// TIA Portal V17 export
// export: Created 2025-03-20T13:42:24.3273325Z, ExportSetting WithDefaults, DisplayName Totally Integrated Automation Portal, DisplayVersion V17 Update 8, DisplayName TIA Portal Openness, DisplayVersion V17 Update 8, DisplayName TIA Portal Version Control Interface, DisplayVersion V17, DisplayName SINAMICS Startdrive Advanced, DisplayVersion V17 SP2, DisplayName SINAMICS Startdrive G110M, G120, G120C, G120D, G120P, G115D, DisplayVersion V17 SP2, DisplayName SINAMICS Startdrive G130, G150, S120, S150, SINAMICS MV, S210, DisplayVersion V17 SP2, DisplayName STEP 7 Professional, DisplayVersion V17 Update 8, DisplayName SINUMERIK ONE STEP 7 Toolbox, DisplayVersion V17 Update 12, DisplayName SINUMERIK 840D sl STEP 7 Toolbox, DisplayVersion V17 Update 12, DisplayName STEP 7 Safety, DisplayVersion V17 Update 6, DisplayName WinCC Advanced, DisplayVersion V17 Update 8
FUNCTION_BLOCK "FB22103_POWDER_LEVEL_SENSOR"   // FB22103, LAD
TITLE = FB22103 CAPACITIVE SENSOR
{ S7_Optimized_Access := 'FALSE' }
VERSION : 0.1
// stored: AutoNumber false, IsIECCheckEnabled false, SetENOAutomatically false, UDAEnableTagReadback false
   VAR_INPUT
      iLOW_LEVEL_SENSOR : Bool;   // LOW LEVEL SENSOR INPUT
      iHIGH_LEVEL_SENSOR : Bool;   // HIGH LEVEL SENSOR INPUT
      iCLEAR_LOG : Bool;   // CLEAR LOG INPUT
   END_VAR
   VAR_OUTPUT
      oLOW_LEVEL_WRN : Bool;   // LOW LEVEL WARNING
      "oHIGH LEVEL_WRN" : Bool;   // HIGH LEVEL WARNING
   END_VAR
   VAR DB_SPECIFIC
      OUTPUT : Struct
         DIGITAL_OUTPUT : Bool;
      END_STRUCT;
      INPUT_SETTINGS : Struct
         UNIT_NUMBER : Int;   // UNIT NUMBER
         HOPPER_NUMBER : Int;   // HOPPER NUMBER
      END_STRUCT;
      ALARMS : Struct   // ALARMS AND WARNINGS
         SENSOR_DISCORDANCY_ALM : Bool;   // SENSOR DISCORDANCY ALARM
      END_STRUCT;
      LOG : Struct
         LAST_EDGE_LOW_LVL : Date_And_Time;   // LAST EDGE LOW LEVEL
         LAST_EDGE_HIGH_LVL : Date_And_Time;   // LAST EDGE HIGH LEVEL
      END_STRUCT;
      INTERNAL : Struct
         RET_VAL : Int;
         AUX1 : Bool;
         AUX2 : Bool;
      END_STRUCT;
   END_VAR
   VAR_TEMP
      DB_NUMBER : DInt;
   END_VAR
   VAR_TEMP   // added for the SCL form of the ladder/FBD networks
      _w1 : Bool;
   END_VAR
BEGIN

NETWORK
TITLE = READ INSTANCE DB NUMBER
      L     DINO;
      +     10#800000;
      T     #DB_NUMBER;

REGION Network 2: LOG LAST EDGE LOW LEVEL (DATE AND TIME)
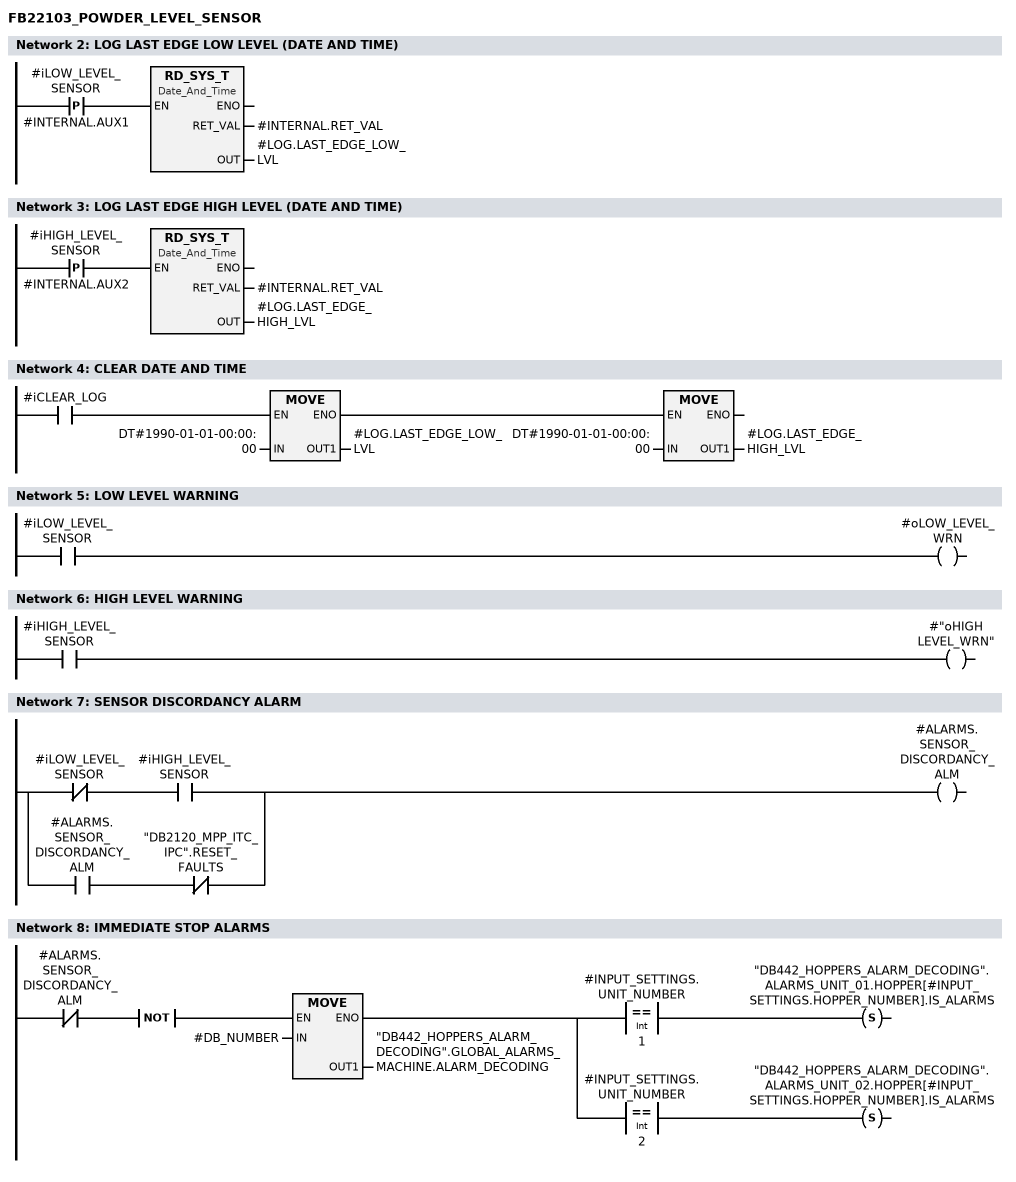
   RUNG wire#powerrail
      P_Contact(operand := #iLOW_LEVEL_SENSOR, bit := #INTERNAL.AUX1)
      { S7_Templates := "date_type := Date_And_Time" } RD_SYS_T(RET_VAL => #INTERNAL.RET_VAL, OUT => #LOG.LAST_EDGE_LOW_LVL)
   END_RUNG
   // the same network as SCL:
   #_w1 := #iLOW_LEVEL_SENSOR AND NOT #INTERNAL.AUX1;   // rising edge of #iLOW_LEVEL_SENSOR
   #INTERNAL.AUX1 := #iLOW_LEVEL_SENSOR;
   IF #_w1 THEN #INTERNAL.RET_VAL := RD_SYS_T(OUT => #LOG.LAST_EDGE_LOW_LVL); END_IF;
END_REGION

REGION Network 3: LOG LAST EDGE HIGH LEVEL (DATE AND TIME)
   RUNG wire#powerrail
      P_Contact(operand := #iHIGH_LEVEL_SENSOR, bit := #INTERNAL.AUX2)
      { S7_Templates := "date_type := Date_And_Time" } RD_SYS_T(RET_VAL => #INTERNAL.RET_VAL, OUT => #LOG.LAST_EDGE_HIGH_LVL)
   END_RUNG
   // the same network as SCL:
   #_w1 := #iHIGH_LEVEL_SENSOR AND NOT #INTERNAL.AUX2;   // rising edge of #iHIGH_LEVEL_SENSOR
   #INTERNAL.AUX2 := #iHIGH_LEVEL_SENSOR;
   IF #_w1 THEN #INTERNAL.RET_VAL := RD_SYS_T(OUT => #LOG.LAST_EDGE_HIGH_LVL); END_IF;
END_REGION

REGION Network 4: CLEAR DATE AND TIME
   RUNG wire#powerrail
      Contact( #iCLEAR_LOG )
      Move(in := DT#1990-01-01-00:00:00, out1 => #LOG.LAST_EDGE_LOW_LVL)
      Move(in := DT#1990-01-01-00:00:00, out1 => #LOG.LAST_EDGE_HIGH_LVL)
   END_RUNG
   // the same network as SCL:
   IF #iCLEAR_LOG THEN
       #LOG.LAST_EDGE_LOW_LVL := DT#1990-01-01-00:00:00;
       #LOG.LAST_EDGE_HIGH_LVL := DT#1990-01-01-00:00:00;
   END_IF;
END_REGION

REGION Network 5: LOW LEVEL WARNING
   RUNG wire#powerrail
      Contact( #iLOW_LEVEL_SENSOR )
      Coil( #oLOW_LEVEL_WRN )
   END_RUNG
   // the same network as SCL:
   #oLOW_LEVEL_WRN := #iLOW_LEVEL_SENSOR;
END_REGION

REGION Network 6: HIGH LEVEL WARNING
   RUNG wire#powerrail
      Contact( #iHIGH_LEVEL_SENSOR )
      Coil( #"oHIGH LEVEL_WRN" )
   END_RUNG
   // the same network as SCL:
   #"oHIGH LEVEL_WRN" := #iHIGH_LEVEL_SENSOR;
END_REGION

REGION Network 7: SENSOR DISCORDANCY ALARM
   RUNG wire#powerrail
      I_Contact( #iLOW_LEVEL_SENSOR )
      Contact( #iHIGH_LEVEL_SENSOR )
      wire#w1
      Coil( #ALARMS.SENSOR_DISCORDANCY_ALM )
   END_RUNG
   RUNG wire#powerrail
      Contact( #ALARMS.SENSOR_DISCORDANCY_ALM )
      I_Contact( "DB2120_MPP_ITC_IPC".RESET_FAULTS )
   END_RUNG wire#w1
   // the same network as SCL:
   #ALARMS.SENSOR_DISCORDANCY_ALM := (NOT #iLOW_LEVEL_SENSOR AND #iHIGH_LEVEL_SENSOR) OR (#ALARMS.SENSOR_DISCORDANCY_ALM AND NOT "DB2120_MPP_ITC_IPC".RESET_FAULTS);
END_REGION

REGION Network 8: IMMEDIATE STOP ALARMS
   RUNG wire#powerrail
      I_Contact( #ALARMS.SENSOR_DISCORDANCY_ALM )
      Not()
      { S7_GenerateENO := "TRUE" } Move(in := #DB_NUMBER, out1 => "DB442_HOPPERS_ALARM_DECODING".GLOBAL_ALARMS_MACHINE.ALARM_DECODING)
      wire#w1
      { S7_Templates := "SrcType := Int" } EQ_Contact(in1 := #INPUT_SETTINGS.UNIT_NUMBER, in2 := 1)
      S_Coil( "DB442_HOPPERS_ALARM_DECODING".ALARMS_UNIT_01.HOPPER[#INPUT_SETTINGS.HOPPER_NUMBER].IS_ALARMS )
   END_RUNG
   RUNG wire#w1
      { S7_Templates := "SrcType := Int" } EQ_Contact(in1 := #INPUT_SETTINGS.UNIT_NUMBER, in2 := 2)
      S_Coil( "DB442_HOPPERS_ALARM_DECODING".ALARMS_UNIT_02.HOPPER[#INPUT_SETTINGS.HOPPER_NUMBER].IS_ALARMS )
   END_RUNG
   // the same network as SCL:
   // ENO of a box is taken as its EN; it also drops when the box reports an error
   #_w1 := NOT (NOT #ALARMS.SENSOR_DISCORDANCY_ALM);
   IF #_w1 THEN "DB442_HOPPERS_ALARM_DECODING".GLOBAL_ALARMS_MACHINE.ALARM_DECODING := #DB_NUMBER; END_IF;
   IF #_w1 AND (#INPUT_SETTINGS.UNIT_NUMBER = 1) THEN
       "DB442_HOPPERS_ALARM_DECODING".ALARMS_UNIT_01.HOPPER[#INPUT_SETTINGS.HOPPER_NUMBER].IS_ALARMS := TRUE;
   END_IF;
   IF #_w1 AND (#INPUT_SETTINGS.UNIT_NUMBER = 2) THEN
       "DB442_HOPPERS_ALARM_DECODING".ALARMS_UNIT_02.HOPPER[#INPUT_SETTINGS.HOPPER_NUMBER].IS_ALARMS := TRUE;
   END_IF;
END_REGION
END_FUNCTION_BLOCK
